PROGRAM PRG_QuestarMotors
VAR
	fbQSTX_Motor : FB_MotionStage;
    fbQSTY_Motor : FB_MotionStage;
END_VAR

Main.M12.bHardwareEnable := TRUE;
fbQSTX_Motor(stMotionStage:=Main.M12);

Main.M13.bHardwareEnable := TRUE;
fbQSTY_Motor(stMotionStage:=Main.M13);

END_PROGRAM

(* stored: Version 1.1.0.1, ProductVersion 3.1.4024.6
   POU PRG_QuestarMotors: Id {b808132d-7d95-489d-997e-88ecb08bbdf8}, SpecialFunc None *)
